LIN {X 0,Y 161.191,Z 829.833,A -85,B 0,C 180,E1 791.183,E2 791.183} C_VEL
LIN {X 0,Y 150.054,Z 833.06,A -85,B 0,C 180,E1 798.079,E2 798.079} C_VEL
LIN {X 0,Y 141.222,Z 834.723,A -85,B 0,C 180,E1 806.347,E2 806.347} C_VEL
LIN {X 0,Y 138.652,Z 835.006,A -85,B 0,C 180,E1 810,E2 810} C_VEL
LIN {X 0,Y 146.048,Z 833.92,A -85,B 0,C 180,E1 818.662,E2 818.662} C_VEL
LIN {X 0,Y 156.674,Z 831.282,A -85,B 0,C 180,E1 826.307,E2 826.307} C_VEL
LIN {X 0,Y 169.142,Z 827.053,A -85,B 0,C 180,E1 832.596,E2 832.596} C_VEL
LIN {X 0,Y 184.047,Z 820.874,A -85,B 0,C 180,E1 838.205,E2 838.205} C_VEL
LIN {X 0,Y 199.626,Z 812.797,A -85,B 0,C 180,E1 842.746,E2 842.746} C_VEL
LIN {X 0,Y 214.601,Z 803.444,A -85,B 0,C 180,E1 846.277,E2 846.277} C_VEL
LIN {X 0,Y 228.557,Z 793.325,A -85,B 0,C 180,E1 849.045,E2 849.045} C_VEL
LIN {X 0,Y 242.092,Z 781.897,A -85,B 0,C 180,E1 851.36,E2 851.36} C_VEL
LIN {X 0,Y 247.393,Z 777.102,A -85,B 0,C 180,E1 852.135,E2 852.135} C_VEL
LIN {X 0,Y 252.833,Z 780.443,A -85,B 0,C 180,E1 847.517,E2 847.517} C_VEL
LIN {X 0,Y 256.814,Z 784.256,A -85,B 0,C 180,E1 842.759,E2 842.759} C_VEL
LIN {X 0,Y 260.866,Z 787.143,A -85,B 0,C 180,E1 838.127,E2 838.127} C_VEL
LIN {X 0,Y 264.812,Z 789.227,A -85,B 0,C 180,E1 833.437,E2 833.437} C_VEL
LIN {X 0,Y 266.278,Z 790.067,A -85,B 0,C 180,E1 831.36,E2 831.36} C_VEL
LIN {X 0,Y 267.886,Z 792.132,A -85,B 0,C 180,E1 827.373,E2 827.373} C_VEL
LIN {X 0,Y 269.552,Z 793.793,A -85,B 0,C 180,E1 823.077,E2 823.077} C_VEL
LIN {X 0,Y 270.707,Z 794.709,A -85,B 0,C 180,E1 819.138,E2 819.138} C_VEL
LIN {X 0,Y 271.558,Z 795.315,A -85,B 0,C 180,E1 815.281,E2 815.281} C_VEL
LIN {X 0,Y 271.962,Z 795.55,A -85,B 0,C 180,E1 811.053,E2 811.053} C_VEL
LIN {X 0,Y 271.858,Z 795.52,A -85,B 0,C 180,E1 807.681,E2 807.681} C_VEL
LIN {X 0,Y 271.419,Z 795.217,A -85,B 0,C 180,E1 804.059,E2 804.059} C_VEL
LIN {X 0,Y 270.446,Z 794.517,A -85,B 0,C 180,E1 799.778,E2 799.778} C_VEL
LIN {X 0,Y 269.206,Z 793.489,A -85,B 0,C 180,E1 796.03,E2 796.03} C_VEL
LIN {X 0,Y 267.647,Z 791.823,A -85,B 0,C 180,E1 791.937,E2 791.937} C_VEL
LIN {X 0,Y 265.93,Z 789.706,A -85,B 0,C 180,E1 787.915,E2 787.915} C_VEL
LIN {X 0,Y 262.307,Z 787.956,A -85,B 0,C 180,E1 783.607,E2 783.607} C_VEL
LIN {X 0,Y 258.761,Z 785.748,A -85,B 0,C 180,E1 779.505,E2 779.505} C_VEL
LIN {X 0,Y 254.938,Z 782.621,A -85,B 0,C 180,E1 775.054,E2 775.054} C_VEL
LIN {X 0,Y 252.057,Z 779.941,A -85,B 0,C 180,E1 771.771,E2 771.771} C_VEL
LIN {X 0,Y 248.404,Z 777.777,A -85,B 0,C 180,E1 768.699,E2 768.699} C_VEL
LIN {X 0,Y 247.692,Z 778.389,A -85,B 0,C 180,E1 768.769,E2 768.769} C_VEL
LIN {X 0,Y 246.801,Z 780.179,A -85,B 0,C 180,E1 769.512,E2 769.512} C_VEL
LIN {X 0,Y 246.581,Z 782.647,A -85,B 0,C 180,E1 771.029,E2 771.029} C_VEL
LIN {X 0,Y 248.589,Z 787.362,A -85,B 0,C 180,E1 775.274,E2 775.274} C_VEL
LIN {X 0,Y 249.614,Z 788.309,A -85,B 0,C 180,E1 776.564,E2 776.564} C_VEL
LIN {X 0,Y 253.438,Z 791.181,A -85,B 0,C 180,E1 780.972,E2 780.972} C_VEL
LIN {X 0,Y 257.537,Z 793.504,A -85,B 0,C 180,E1 785.7,E2 785.7} C_VEL
LIN {X 0,Y 259.769,Z 794.706,A -85,B 0,C 180,E1 788.664,E2 788.664} C_VEL
LIN {X 0,Y 261.47,Z 796.876,A -85,B 0,C 180,E1 792.876,E2 792.876} C_VEL
LIN {X 0,Y 263.104,Z 798.46,A -85,B 0,C 180,E1 797.267,E2 797.267} C_VEL
LIN {X 0,Y 264.265,Z 799.389,A -85,B 0,C 180,E1 801.296,E2 801.296} C_VEL
LIN {X 0,Y 265.054,Z 799.949,A -85,B 0,C 180,E1 805.023,E2 805.023} C_VEL
LIN {X 0,Y 265.506,Z 800.23,A -85,B 0,C 180,E1 809.137,E2 809.137} C_VEL
LIN {X 0,Y 265.278,Z 800.09,A -85,B 0,C 180,E1 813.241,E2 813.241} C_VEL
LIN {X 0,Y 264.726,Z 799.721,A -85,B 0,C 180,E1 816.724,E2 816.724} C_VEL
LIN {X 0,Y 263.677,Z 798.965,A -85,B 0,C 180,E1 820.929,E2 820.929} C_VEL
LIN {X 0,Y 262.186,Z 797.59,A -85,B 0,C 180,E1 825.256,E2 825.256} C_VEL
LIN {X 0,Y 260.721,Z 795.948,A -85,B 0,C 180,E1 829.024,E2 829.024} C_VEL
LIN {X 0,Y 259.221,Z 794.266,A -85,B 0,C 180,E1 832.223,E2 832.223} C_VEL
LIN {X 0,Y 255.874,Z 792.651,A -85,B 0,C 180,E1 836.203,E2 836.203} C_VEL
LIN {X 0,Y 252.068,Z 790.252,A -85,B 0,C 180,E1 840.599,E2 840.599} C_VEL
LIN {X 0,Y 247.848,Z 786.686,A -85,B 0,C 180,E1 845.514,E2 845.514} C_VEL
LIN {X 0,Y 245.758,Z 784.692,A -85,B 0,C 180,E1 847.903,E2 847.903} C_VEL
LIN {X 0,Y 243.842,Z 783.834,A -85,B 0,C 180,E1 849.351,E2 849.351} C_VEL
LIN {X 0,Y 230.139,Z 795.416,A -85,B 0,C 180,E1 846.837,E2 846.837} C_VEL
LIN {X 0,Y 214.56,Z 806.667,A -85,B 0,C 180,E1 843.473,E2 843.473} C_VEL
LIN {X 0,Y 199.974,Z 815.591,A -85,B 0,C 180,E1 839.668,E2 839.668} C_VEL
LIN {X 0,Y 187.268,Z 822.116,A -85,B 0,C 180,E1 835.624,E2 835.624} C_VEL
LIN {X 0,Y 174.366,Z 827.654,A -85,B 0,C 180,E1 830.474,E2 830.474} C_VEL
LIN {X 0,Y 161.473,Z 831.902,A -85,B 0,C 180,E1 823.552,E2 823.552} C_VEL
LIN {X 0,Y 152.275,Z 834.072,A -85,B 0,C 180,E1 816.409,E2 816.409} C_VEL
LIN {X 0,Y 146.979,Z 834.745,A -85,B 0,C 180,E1 809.873,E2 809.873} C_VEL
LIN {X 0,Y 154.243,Z 833.662,A -85,B 0,C 180,E1 801.801,E2 801.801} C_VEL
LIN {X 0,Y 164.654,Z 831.022,A -85,B 0,C 180,E1 794.503,E2 794.503} C_VEL
LIN {X 0,Y 177.456,Z 826.447,A -85,B 0,C 180,E1 788.17,E2 788.17} C_VEL
LIN {X 0,Y 191.393,Z 820.154,A -85,B 0,C 180,E1 782.968,E2 782.968} C_VEL
LIN {X 0,Y 206.646,Z 811.717,A -85,B 0,C 180,E1 778.497,E2 778.497} C_VEL
LIN {X 0,Y 220.535,Z 802.577,A -85,B 0,C 180,E1 775.163,E2 775.163} C_VEL
LIN {X 0,Y 235.031,Z 791.492,A -85,B 0,C 180,E1 772.224,E2 772.224} C_VEL
LIN {X 0,Y 244.056,Z 783.74,A -85,B 0,C 180,E1 770.648,E2 770.648} C_VEL
LIN {X 0,Y 246.647,Z 785.425,A -85,B 0,C 180,E1 772.996,E2 772.996} C_VEL
LIN {X 0,Y 249.614,Z 788.309,A -85,B 0,C 180,E1 776.564,E2 776.564} C_VEL
LIN {X 0,Y 250.287,Z 790.07,A -85,B 0,C 180,E1 778.29,E2 778.29} C_VEL
LIN {X 0,Y 249.306,Z 794.473,A -85,B 0,C 180,E1 781.47,E2 781.47} C_VEL
LIN {X 0,Y 249.24,Z 796.903,A -85,B 0,C 180,E1 783.724,E2 783.724} C_VEL
LIN {X 0,Y 249.7,Z 797.308,A -85,B 0,C 180,E1 784.481,E2 784.481} C_VEL
LIN {X 0,Y 252.985,Z 798.955,A -85,B 0,C 180,E1 788.436,E2 788.436} C_VEL
LIN {X 0,Y 254.531,Z 800.946,A -85,B 0,C 180,E1 792.394,E2 792.394} C_VEL
LIN {X 0,Y 256.249,Z 802.702,A -85,B 0,C 180,E1 796.92,E2 796.92} C_VEL
LIN {X 0,Y 257.515,Z 803.726,A -85,B 0,C 180,E1 801.066,E2 801.066} C_VEL
LIN {X 0,Y 258.293,Z 804.265,A -85,B 0,C 180,E1 804.669,E2 804.669} C_VEL
LIN {X 0,Y 258.765,Z 804.576,A -85,B 0,C 180,E1 808.893,E2 808.893} C_VEL
LIN {X 0,Y 258.575,Z 804.451,A -85,B 0,C 180,E1 813.103,E2 813.103} C_VEL
LIN {X 0,Y 258.041,Z 804.11,A -85,B 0,C 180,E1 816.675,E2 816.675} C_VEL
LIN {X 0,Y 257.068,Z 803.379,A -85,B 0,C 180,E1 820.533,E2 820.533} C_VEL
LIN {X 0,Y 255.551,Z 802.014,A -85,B 0,C 180,E1 824.965,E2 824.965} C_VEL
LIN {X 0,Y 253.888,Z 800.156,A -85,B 0,C 180,E1 829.317,E2 829.317} C_VEL
LIN {X 0,Y 252.543,Z 798.664,A -85,B 0,C 180,E1 832.114,E2 832.114} C_VEL
LIN {X 0,Y 248.628,Z 796.725,A -85,B 0,C 180,E1 836.777,E2 836.777} C_VEL
LIN {X 0,Y 244.208,Z 793.726,A -85,B 0,C 180,E1 841.88,E2 841.88} C_VEL
LIN {X 0,Y 240.29,Z 790.365,A -85,B 0,C 180,E1 846.328,E2 846.328} C_VEL
LIN {X 0,Y 224.276,Z 803.023,A -85,B 0,C 180,E1 842.948,E2 842.948} C_VEL
LIN {X 0,Y 209.362,Z 813.06,A -85,B 0,C 180,E1 839.151,E2 839.151} C_VEL
LIN {X 0,Y 195.439,Z 820.831,A -85,B 0,C 180,E1 834.803,E2 834.803} C_VEL
LIN {X 0,Y 182.758,Z 826.742,A -85,B 0,C 180,E1 829.827,E2 829.827} C_VEL
LIN {X 0,Y 170.823,Z 831.189,A -85,B 0,C 180,E1 823.681,E2 823.681} C_VEL
LIN {X 0,Y 161.266,Z 833.648,A -85,B 0,C 180,E1 816.765,E2 816.765} C_VEL
LIN {X 0,Y 155.145,Z 834.494,A -85,B 0,C 180,E1 810,E2 810} C_VEL
LIN {X 0,Y 162.047,Z 833.475,A -85,B 0,C 180,E1 802.555,E2 802.555} C_VEL
LIN {X 0,Y 171.631,Z 830.924,A -85,B 0,C 180,E1 795.838,E2 795.838} C_VEL
LIN {X 0,Y 183.964,Z 826.27,A -85,B 0,C 180,E1 789.645,E2 789.645} C_VEL
LIN {X 0,Y 197.451,Z 819.832,A -85,B 0,C 180,E1 784.506,E2 784.506} C_VEL
LIN {X 0,Y 211.54,Z 811.666,A -85,B 0,C 180,E1 780.246,E2 780.246} C_VEL
LIN {X 0,Y 226.591,Z 801.374,A -85,B 0,C 180,E1 776.526,E2 776.526} C_VEL
LIN {X 0,Y 240.444,Z 790.318,A -85,B 0,C 180,E1 773.679,E2 773.679} C_VEL
LIN {X 0,Y 244.965,Z 794.309,A -85,B 0,C 180,E1 778.997,E2 778.997} C_VEL
LIN {X 0,Y 249.273,Z 797.096,A -85,B 0,C 180,E1 783.959,E2 783.959} C_VEL
LIN {X 0,Y 249.7,Z 797.308,A -85,B 0,C 180,E1 784.481,E2 784.481} C_VEL
LIN {X 0,Y 250.225,Z 798.546,A -85,B 0,C 180,E1 786.107,E2 786.107} C_VEL
LIN {X 0,Y 249.124,Z 801.247,A -85,B 0,C 180,E1 788.456,E2 788.456} C_VEL
LIN {X 0,Y 247.551,Z 804.441,A -85,B 0,C 180,E1 791.492,E2 791.492} C_VEL
LIN {X 0,Y 247.685,Z 805.064,A -85,B 0,C 180,E1 792.528,E2 792.528} C_VEL
LIN {X 0,Y 249.404,Z 806.82,A -85,B 0,C 180,E1 797.027,E2 797.027} C_VEL
LIN {X 0,Y 250.593,Z 807.746,A -85,B 0,C 180,E1 801.048,E2 801.048} C_VEL
LIN {X 0,Y 251.39,Z 808.298,A -85,B 0,C 180,E1 804.751,E2 804.751} C_VEL
LIN {X 0,Y 251.872,Z 808.605,A -85,B 0,C 180,E1 809.09,E2 809.09} C_VEL
LIN {X 0,Y 251.656,Z 808.474,A -85,B 0,C 180,E1 813.189,E2 813.189} C_VEL
LIN {X 0,Y 251.083,Z 808.088,A -85,B 0,C 180,E1 816.861,E2 816.861} C_VEL
LIN {X 0,Y 250.019,Z 807.343,A -85,B 0,C 180,E1 821.067,E2 821.067} C_VEL
LIN {X 0,Y 248.505,Z 805.928,A -85,B 0,C 180,E1 825.399,E2 825.399} C_VEL
LIN {X 0,Y 246.723,Z 803.884,A -85,B 0,C 180,E1 829.917,E2 829.917} C_VEL
LIN {X 0,Y 245.73,Z 802.835,A -85,B 0,C 180,E1 831.983,E2 831.983} C_VEL
LIN {X 0,Y 242.046,Z 800.97,A -85,B 0,C 180,E1 836.312,E2 836.312} C_VEL
LIN {X 0,Y 238.249,Z 798.481,A -85,B 0,C 180,E1 840.648,E2 840.648} C_VEL
LIN {X 0,Y 236.285,Z 796.981,A -85,B 0,C 180,E1 842.981,E2 842.981} C_VEL
LIN {X 0,Y 220.906,Z 808.433,A -85,B 0,C 180,E1 839.263,E2 839.263} C_VEL
LIN {X 0,Y 206.114,Z 817.688,A -85,B 0,C 180,E1 834.888,E2 834.888} C_VEL
LIN {X 0,Y 194.148,Z 824.084,A -85,B 0,C 180,E1 830.499,E2 830.499} C_VEL
LIN {X 0,Y 182.244,Z 829.205,A -85,B 0,C 180,E1 824.943,E2 824.943} C_VEL
LIN {X 0,Y 172.293,Z 832.49,A -85,B 0,C 180,E1 818.678,E2 818.678} C_VEL
LIN {X 0,Y 165.06,Z 834.011,A -85,B 0,C 180,E1 812.083,E2 812.083} C_VEL
LIN {X 0,Y 163.394,Z 834.158,A -85,B 0,C 180,E1 810,E2 810} C_VEL
LIN {X 0,Y 170.28,Z 833.024,A -85,B 0,C 180,E1 802.903,E2 802.903} C_VEL
LIN {X 0,Y 180.183,Z 829.999,A -85,B 0,C 180,E1 796.196,E2 796.196} C_VEL
LIN {X 0,Y 192.221,Z 824.998,A -85,B 0,C 180,E1 790.303,E2 790.303} C_VEL
LIN {X 0,Y 204.948,Z 818.429,A -85,B 0,C 180,E1 785.501,E2 785.501} C_VEL
LIN {X 0,Y 220.185,Z 808.954,A -85,B 0,C 180,E1 780.93,E2 780.93} C_VEL
LIN {X 0,Y 235.784,Z 797.354,A -85,B 0,C 180,E1 777.127,E2 777.127} C_VEL
LIN {X 0,Y 236.278,Z 796.954,A -85,B 0,C 180,E1 777.019,E2 777.019} C_VEL
LIN {X 0,Y 240.869,Z 800.273,A -85,B 0,C 180,E1 782.296,E2 782.296} C_VEL
LIN {X 0,Y 245.092,Z 802.566,A -85,B 0,C 180,E1 787.216,E2 787.216} C_VEL
LIN {X 0,Y 246.326,Z 803.351,A -85,B 0,C 180,E1 789.072,E2 789.072} C_VEL
LIN {X 0,Y 247.685,Z 805.064,A -85,B 0,C 180,E1 792.528,E2 792.528} C_VEL
LIN {X 0,Y 247.513,Z 806.334,A -85,B 0,C 180,E1 794.299,E2 794.299} C_VEL
LIN {X 0,Y 245.132,Z 809.166,A -85,B 0,C 180,E1 797.171,E2 797.171} C_VEL
LIN {X 0,Y 243.419,Z 811.206,A -85,B 0,C 180,E1 799.874,E2 799.874} C_VEL
LIN {X 0,Y 243.44,Z 811.431,A -85,B 0,C 180,E1 800.665,E2 800.665} C_VEL
LIN {X 0,Y 244.271,Z 812.05,A -85,B 0,C 180,E1 804.362,E2 804.362} C_VEL
LIN {X 0,Y 244.779,Z 812.421,A -85,B 0,C 180,E1 808.596,E2 808.596} C_VEL
LIN {X 0,Y 244.662,Z 812.333,A -85,B 0,C 180,E1 812.811,E2 812.811} C_VEL
LIN {X 0,Y 244.084,Z 811.922,A -85,B 0,C 180,E1 816.586,E2 816.586} C_VEL
LIN {X 0,Y 243.077,Z 811.165,A -85,B 0,C 180,E1 820.553,E2 820.553} C_VEL
LIN {X 0,Y 241.581,Z 809.861,A -85,B 0,C 180,E1 825.114,E2 825.114} C_VEL
LIN {X 0,Y 239.845,Z 807.876,A -85,B 0,C 180,E1 829.481,E2 829.481} C_VEL
LIN {X 0,Y 238.682,Z 806.653,A -85,B 0,C 180,E1 831.89,E2 831.89} C_VEL
LIN {X 0,Y 235.72,Z 805.199,A -85,B 0,C 180,E1 835.38,E2 835.38} C_VEL
LIN {X 0,Y 232.219,Z 803.128,A -85,B 0,C 180,E1 839.331,E2 839.331} C_VEL
LIN {X 0,Y 218.424,Z 812.906,A -85,B 0,C 180,E1 835.485,E2 835.485} C_VEL
LIN {X 0,Y 206.133,Z 820.202,A -85,B 0,C 180,E1 831.333,E2 831.333} C_VEL
LIN {X 0,Y 195.03,Z 825.976,A -85,B 0,C 180,E1 826.684,E2 826.684} C_VEL
LIN {X 0,Y 184.858,Z 830.161,A -85,B 0,C 180,E1 821.228,E2 821.228} C_VEL
LIN {X 0,Y 175.898,Z 832.876,A -85,B 0,C 180,E1 814.564,E2 814.564} C_VEL
LIN {X 0,Y 171.629,Z 833.562,A -85,B 0,C 180,E1 810,E2 810} C_VEL
LIN {X 0,Y 178.469,Z 832.21,A -85,B 0,C 180,E1 803.244,E2 803.244} C_VEL
LIN {X 0,Y 187.732,Z 829.107,A -85,B 0,C 180,E1 797.073,E2 797.073} C_VEL
LIN {X 0,Y 198.969,Z 824.082,A -85,B 0,C 180,E1 791.544,E2 791.544} C_VEL
LIN {X 0,Y 212.47,Z 816.626,A -85,B 0,C 180,E1 786.423,E2 786.423} C_VEL
LIN {X 0,Y 225.603,Z 807.981,A -85,B 0,C 180,E1 782.422,E2 782.422} C_VEL
LIN {X 0,Y 232.329,Z 803.133,A -85,B 0,C 180,E1 780.701,E2 780.701} C_VEL
LIN {X 0,Y 236.558,Z 805.675,A -85,B 0,C 180,E1 785.531,E2 785.531} C_VEL
LIN {X 0,Y 239.216,Z 807.047,A -85,B 0,C 180,E1 788.934,E2 788.934} C_VEL
LIN {X 0,Y 241.095,Z 809.389,A -85,B 0,C 180,E1 793.62,E2 793.62} C_VEL
LIN {X 0,Y 242.593,Z 810.751,A -85,B 0,C 180,E1 797.866,E2 797.866} C_VEL
LIN {X 0,Y 243.44,Z 811.431,A -85,B 0,C 180,E1 800.665,E2 800.665} C_VEL
LIN {X 0,Y 243.035,Z 812.235,A -85,B 0,C 180,E1 802.351,E2 802.351} C_VEL
LIN {X 0,Y 240.392,Z 814.139,A -85,B 0,C 180,E1 805.028,E2 805.028} C_VEL
LIN {X 0,Y 237.834,Z 815.797,A -85,B 0,C 180,E1 807.914,E2 807.914} C_VEL
LIN {X 0,Y 237.642,Z 815.944,A -85,B 0,C 180,E1 808.996,E2 808.996} C_VEL
LIN {X 0,Y 237.446,Z 815.822,A -85,B 0,C 180,E1 813.138,E2 813.138} C_VEL
LIN {X 0,Y 236.838,Z 815.403,A -85,B 0,C 180,E1 817.032,E2 817.032} C_VEL
LIN {X 0,Y 235.681,Z 814.522,A -85,B 0,C 180,E1 821.253,E2 821.253} C_VEL
LIN {X 0,Y 234.003,Z 812.966,A -85,B 0,C 180,E1 825.974,E2 825.974} C_VEL
LIN {X 0,Y 232.349,Z 811.028,A -85,B 0,C 180,E1 830.264,E2 830.264} C_VEL
LIN {X 0,Y 231.258,Z 810.134,A -85,B 0,C 180,E1 832.095,E2 832.095} C_VEL
LIN {X 0,Y 228.322,Z 808.816,A -85,B 0,C 180,E1 835.344,E2 835.344} C_VEL
LIN {X 0,Y 215.51,Z 817.229,A -85,B 0,C 180,E1 831.166,E2 831.166} C_VEL
LIN {X 0,Y 206.771,Z 822.252,A -85,B 0,C 180,E1 827.736,E2 827.736} C_VEL
LIN {X 0,Y 194.8,Z 828.043,A -85,B 0,C 180,E1 821.847,E2 821.847} C_VEL
LIN {X 0,Y 185.899,Z 831.321,A -85,B 0,C 180,E1 815.865,E2 815.865} C_VEL
LIN {X 0,Y 179.85,Z 832.652,A -85,B 0,C 180,E1 810,E2 810} C_VEL
LIN {X 0,Y 186.647,Z 831.048,A -85,B 0,C 180,E1 803.541,E2 803.541} C_VEL
LIN {X 0,Y 195.763,Z 827.666,A -85,B 0,C 180,E1 797.613,E2 797.613} C_VEL
LIN {X 0,Y 207.342,Z 821.985,A -85,B 0,C 180,E1 792.024,E2 792.024} C_VEL
LIN {X 0,Y 219.36,Z 814.852,A -85,B 0,C 180,E1 787.489,E2 787.489} C_VEL
LIN {X 0,Y 228.496,Z 808.756,A -85,B 0,C 180,E1 784.636,E2 784.636} C_VEL
LIN {X 0,Y 231.976,Z 810.496,A -85,B 0,C 180,E1 788.774,E2 788.774} C_VEL
LIN {X 0,Y 233.761,Z 812.72,A -85,B 0,C 180,E1 793.356,E2 793.356} C_VEL
LIN {X 0,Y 235.349,Z 814.215,A -85,B 0,C 180,E1 797.736,E2 797.736} C_VEL
LIN {X 0,Y 236.688,Z 815.344,A -85,B 0,C 180,E1 802.231,E2 802.231} C_VEL
LIN {X 0,Y 237.431,Z 815.804,A -85,B 0,C 180,E1 806.62,E2 806.62} C_VEL
LIN {X 0,Y 237.642,Z 815.944,A -85,B 0,C 180,E1 808.996,E2 808.996} C_VEL
LIN {X 0,Y 236.928,Z 816.255,A -85,B 0,C 180,E1 810.721,E2 810.721} C_VEL
LIN {X 0,Y 233.9,Z 817.386,A -85,B 0,C 180,E1 813.183,E2 813.183} C_VEL
LIN {X 0,Y 230.06,Z 818.519,A -85,B 0,C 180,E1 816.254,E2 816.254} C_VEL
LIN {X 0,Y 229.376,Z 818.483,A -85,B 0,C 180,E1 817.511,E2 817.511} C_VEL
LIN {X 0,Y 228.095,Z 817.56,A -85,B 0,C 180,E1 822.171,E2 822.171} C_VEL
LIN {X 0,Y 226.382,Z 815.874,A -85,B 0,C 180,E1 826.683,E2 826.683} C_VEL
LIN {X 0,Y 224.727,Z 813.841,A -85,B 0,C 180,E1 830.973,E2 830.973} C_VEL
LIN {X 0,Y 215.108,Z 819.781,A -85,B 0,C 180,E1 827.306,E2 827.306} C_VEL
LIN {X 0,Y 204.231,Z 825.613,A -85,B 0,C 180,E1 822.152,E2 822.152} C_VEL
LIN {X 0,Y 194.79,Z 829.574,A -85,B 0,C 180,E1 816.188,E2 816.188} C_VEL
LIN {X 0,Y 188.567,Z 831.299,A -85,B 0,C 180,E1 810.608,E2 810.608} C_VEL
LIN {X 0,Y 188.031,Z 831.403,A -85,B 0,C 180,E1 810,E2 810} C_VEL
LIN {X 0,Y 194.408,Z 829.665,A -85,B 0,C 180,E1 804.096,E2 804.096} C_VEL
LIN {X 0,Y 203.762,Z 825.876,A -85,B 0,C 180,E1 798.107,E2 798.107} C_VEL
LIN {X 0,Y 213.453,Z 820.744,A -85,B 0,C 180,E1 793.398,E2 793.398} C_VEL
LIN {X 0,Y 224.745,Z 813.876,A -85,B 0,C 180,E1 789.019,E2 789.019} C_VEL
LIN {X 0,Y 226.604,Z 816.101,A -85,B 0,C 180,E1 793.861,E2 793.861} C_VEL
LIN {X 0,Y 228.162,Z 817.596,A -85,B 0,C 180,E1 798.114,E2 798.114} C_VEL
LIN {X 0,Y 229.451,Z 818.555,A -85,B 0,C 180,E1 802.74,E2 802.74} C_VEL
LIN {X 0,Y 230.119,Z 818.984,A -85,B 0,C 180,E1 807.011,E2 807.011} C_VEL
LIN {X 0,Y 230.234,Z 819.083,A -85,B 0,C 180,E1 810.498,E2 810.498} C_VEL
LIN {X 0,Y 229.964,Z 818.895,A -85,B 0,C 180,E1 814.239,E2 814.239} C_VEL
LIN {X 0,Y 229.376,Z 818.483,A -85,B 0,C 180,E1 817.511,E2 817.511} C_VEL
LIN {X 0,Y 228.129,Z 818.749,A -85,B 0,C 180,E1 818.773,E2 818.773} C_VEL
LIN {X 0,Y 221.087,Z 820.215,A -85,B 0,C 180,E1 822.2,E2 822.2} C_VEL
LIN {X 0,Y 220.233,Z 820.086,A -85,B 0,C 180,E1 823.155,E2 823.155} C_VEL
LIN {X 0,Y 219.389,Z 819.495,A -85,B 0,C 180,E1 825.192,E2 825.192} C_VEL
LIN {X 0,Y 209.868,Z 824.55,A -85,B 0,C 180,E1 820.43,E2 820.43} C_VEL
LIN {X 0,Y 201.775,Z 828.125,A -85,B 0,C 180,E1 815.116,E2 815.116} C_VEL
LIN {X 0,Y 196.15,Z 829.772,A -85,B 0,C 180,E1 810,E2 810} C_VEL
LIN {X 0,Y 203.25,Z 827.571,A -85,B 0,C 180,E1 803.787,E2 803.787} C_VEL
LIN {X 0,Y 212.172,Z 823.457,A -85,B 0,C 180,E1 798.309,E2 798.309} C_VEL
LIN {X 0,Y 219.527,Z 819.427,A -85,B 0,C 180,E1 794.784,E2 794.784} C_VEL
LIN {X 0,Y 221.12,Z 820.819,A -85,B 0,C 180,E1 799.58,E2 799.58} C_VEL
LIN {X 0,Y 222.179,Z 821.594,A -85,B 0,C 180,E1 803.8,E2 803.8} C_VEL
LIN {X 0,Y 222.712,Z 821.976,A -85,B 0,C 180,E1 807.684,E2 807.684} C_VEL
LIN {X 0,Y 222.804,Z 822.014,A -85,B 0,C 180,E1 811.543,E2 811.543} C_VEL
LIN {X 0,Y 222.215,Z 821.649,A -85,B 0,C 180,E1 816.073,E2 816.073} C_VEL
LIN {X 0,Y 221.11,Z 820.797,A -85,B 0,C 180,E1 820.421,E2 820.421} C_VEL
LIN {X 0,Y 220.233,Z 820.086,A -85,B 0,C 180,E1 823.155,E2 823.155} C_VEL
LIN {X 0,Y 219.185,Z 820.512,A -85,B 0,C 180,E1 823.134,E2 823.134} C_VEL
LIN {X 0,Y 217.019,Z 821.672,A -85,B 0,C 180,E1 822.344,E2 822.344} C_VEL
LIN {X 0,Y 214.463,Z 823.16,A -85,B 0,C 180,E1 820.423,E2 820.423} C_VEL
LIN {X 0,Y 210.499,Z 825.642,A -85,B 0,C 180,E1 815.691,E2 815.691} C_VEL
LIN {X 0,Y 208.845,Z 826.286,A -85,B 0,C 180,E1 814.196,E2 814.196} C_VEL
LIN {X 0,Y 204.215,Z 827.892,A -85,B 0,C 180,E1 810,E2 810} C_VEL
LIN {X 0,Y 211.252,Z 825.311,A -85,B 0,C 180,E1 804.023,E2 804.023} C_VEL
LIN {X 0,Y 214.273,Z 824.037,A -85,B 0,C 180,E1 802.109,E2 802.109} C_VEL
LIN {X 0,Y 215.073,Z 824.55,A -85,B 0,C 180,E1 806.535,E2 806.535} C_VEL
LIN {X 0,Y 215.245,Z 824.67,A -85,B 0,C 180,E1 810.266,E2 810.266} C_VEL
LIN {X 0,Y 214.967,Z 824.483,A -85,B 0,C 180,E1 814.268,E2 814.268} C_VEL
LIN {X 0,Y 214.21,Z 823.99,A -85,B 0,C 180,E1 817.932,E2 817.932} C_VEL
LIN {X 0,Y 208.845,Z 826.286,A -85,B 0,C 180,E1 814.196,E2 814.196} C_VEL
LIN {X 0,Y 208.276,Z 828.27,A -85,B 0,C 180,E1 813.743,E2 813.743} C_VEL
LIN {X 0,Y 208.276,Z 862.5,A -85,B 0,C 180,E1 813.743,E2 813.743} C_VEL
LIN {X 0,Y 208.276,Z 862.5,A -85,B 0,C 180,E1 813.743,E2 813.743}

QRS_NEXT_CUT()

QRS_NEXT()
QRS_HOME()

END
